// TIA Portal project "Lab5_Exp1_PunchingMachine" (V16)

(* hardware
DEVICE "S7300/ET200M station_1"  S7-300 station
   slot 0: "Rail_0"  Rail  6ES7 390-1***0-0AA0
   slot 2: "PLC_1"  CPU 317-2 PN/DP  6ES7 317-2EK14-0AB0  V3.2
      slot 2: "PROFINET interface_1"  PN-IO
         slot 1: "Port_1"  Port
         slot 2: "Port_2"  Port
*)

// ===== PLC "PLC_1"  CPU 317-2 PN/DP =====

VAR_GLOBAL   // PLC tag table "Default tag table"
   "diStartB" AT %I0.1 : Bool;
   "diGuardDown" AT %I0.2 : Bool;
   "diPunchUp" AT %I0.3 : Bool;
   "diPunchDown" AT %I0.4 : Bool;
   "diStopB" AT %I0.5 : Bool;
   "doPunchDown" AT %Q0.0 : Bool;
   "doReadyIndicator" AT %Q0.1 : Bool;
   "doGDIndicator" AT %Q0.3 : Bool;
   "doGuardDown" AT %Q0.4 : Bool;
   "tvDelayT1" AT %QW66 : Word;
   "tvDelayT2" AT %QW68 : Word;
   "mS_Stop" AT %M100.0 : Bool;
   "mS_GuardDown" AT %M100.1 : Bool;
   "mS_PunchDown" AT %M100.2 : Bool;
   "mS_DelayT1" AT %M100.3 : Bool;
   "mS_GuardUp" AT %M100.4 : Bool;
   "mS_PunchUp" AT %M100.5 : Bool;
   "mT1Elapsed" AT %M100.6 : Bool;
   "mT2Elapsed" AT %M100.7 : Bool;
   "DelayT1" AT %T1 : Timer;
   "DelayT2" AT %T2 : Timer;
   "Tag_1" AT %M200.0 : Bool;
END_VAR

ORGANIZATION_BLOCK "Main"   // OB1, LAD
TITLE = "Main Program Sweep (Cycle)"
{ S7_Optimized_Access := 'FALSE' }
VERSION : 0.1
   VAR_TEMP
      OB1_EV_CLASS : Byte;   // Bits 0-3 = 1 (Coming event), Bits 4-7 = 1 (Event class 1)
      OB1_SCAN_1 : Byte;   // 1 (Cold restart scan 1 of OB 1), 3 (Scan 2-n of OB 1)
      OB1_PRIORITY : Byte;   // Priority of OB Execution
      OB1_OB_NUMBR : Byte;   // 1 (Organization block 1, OB1)
      OB1_RESERVED_1 : Byte;   // Reserved for system
      OB1_RESERVED_2 : Byte;   // Reserved for system
      OB1_PREV_CYCLE : Int;   // Cycle time of previous OB1 scan (milliseconds)
      OB1_MIN_CYCLE : Int;   // Minimum cycle time of OB1 (milliseconds)
      OB1_MAX_CYCLE : Int;   // Maximum cycle time of OB1 (milliseconds)
      OB1_DATE_TIME : Date_And_Time;   // Date and time OB1 started
   END_VAR
   VAR_TEMP   // added for the SCL form of the ladder/FBD networks
      _w1 : Bool;
      _s5time1 : S5Time;
   END_VAR
BEGIN

REGION Network 1: Setting mS_Stop
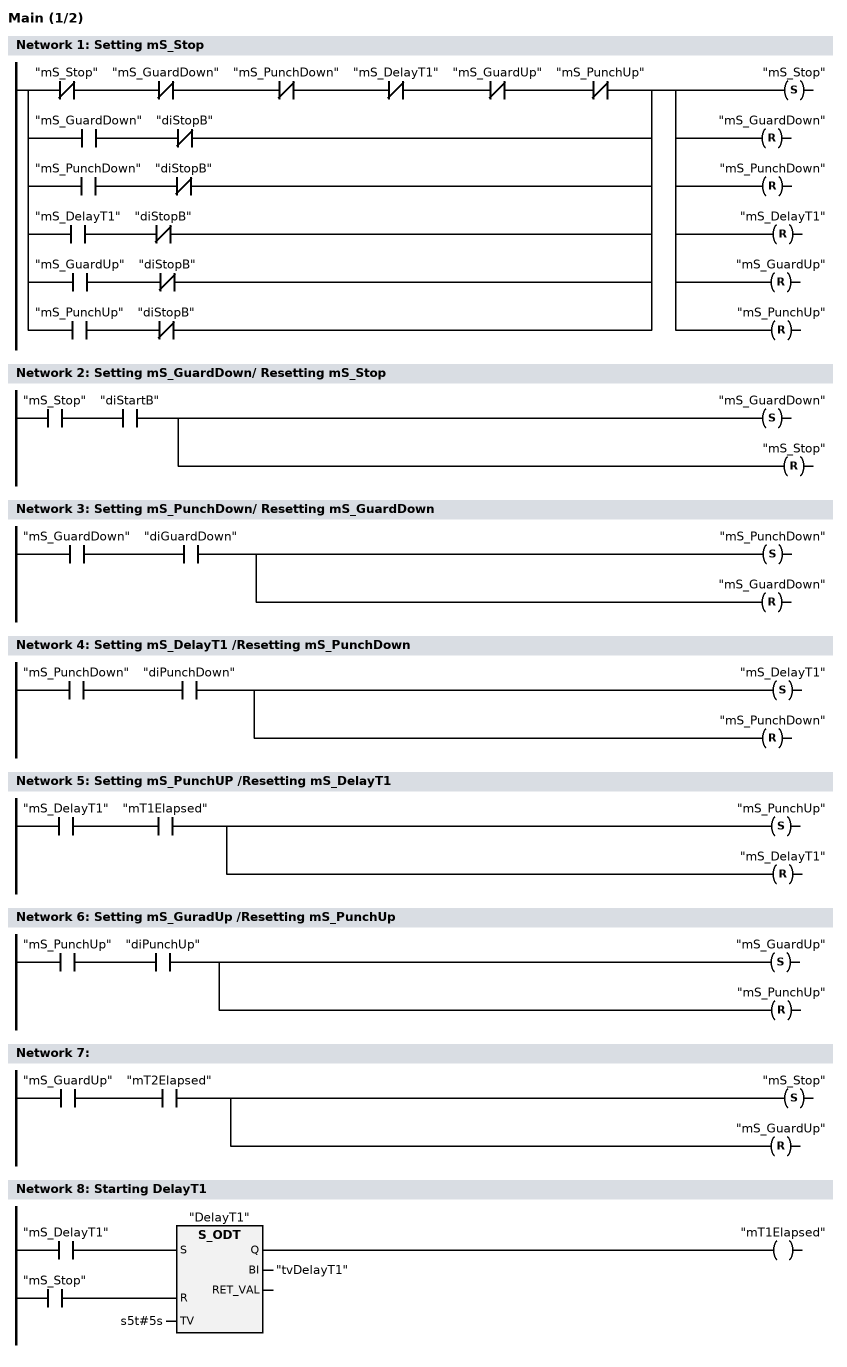
   RUNG wire#powerrail
      I_Contact( "mS_Stop" )
      I_Contact( "mS_GuardDown" )
      I_Contact( "mS_PunchDown" )
      I_Contact( "mS_DelayT1" )
      I_Contact( "mS_GuardUp" )
      I_Contact( "mS_PunchUp" )
      wire#w1
      S_Coil( "mS_Stop" )
   END_RUNG
   RUNG wire#powerrail
      Contact( "mS_GuardDown" )
      I_Contact( "diStopB" )
   END_RUNG wire#w1
   RUNG wire#powerrail
      Contact( "mS_PunchDown" )
      I_Contact( "diStopB" )
   END_RUNG wire#w1
   RUNG wire#powerrail
      Contact( "mS_DelayT1" )
      I_Contact( "diStopB" )
   END_RUNG wire#w1
   RUNG wire#powerrail
      Contact( "mS_GuardUp" )
      I_Contact( "diStopB" )
   END_RUNG wire#w1
   RUNG wire#powerrail
      Contact( "mS_PunchUp" )
      I_Contact( "diStopB" )
   END_RUNG wire#w1
   RUNG wire#w1
      R_Coil( "mS_GuardDown" )
   END_RUNG
   RUNG wire#w1
      R_Coil( "mS_PunchDown" )
   END_RUNG
   RUNG wire#w1
      R_Coil( "mS_DelayT1" )
   END_RUNG
   RUNG wire#w1
      R_Coil( "mS_GuardUp" )
   END_RUNG
   RUNG wire#w1
      R_Coil( "mS_PunchUp" )
   END_RUNG
   // the same network as SCL:
   #_w1 := (NOT "mS_Stop" AND NOT "mS_GuardDown" AND NOT "mS_PunchDown" AND NOT "mS_DelayT1" AND NOT "mS_GuardUp" AND NOT "mS_PunchUp") OR ("mS_GuardDown" AND NOT "diStopB") OR ("mS_PunchDown" AND NOT "diStopB") OR ("mS_DelayT1" AND NOT "diStopB") OR ("mS_GuardUp" AND NOT "diStopB") OR ("mS_PunchUp" AND NOT "diStopB");
   IF #_w1 THEN
       "mS_Stop" := TRUE;
       "mS_GuardDown" := FALSE;
       "mS_PunchDown" := FALSE;
       "mS_DelayT1" := FALSE;
       "mS_GuardUp" := FALSE;
       "mS_PunchUp" := FALSE;
   END_IF;
END_REGION

REGION Network 2: Setting mS_GuardDown/ Resetting mS_Stop
   RUNG wire#powerrail
      Contact( "mS_Stop" )
      Contact( "diStartB" )
      wire#w1
      S_Coil( "mS_GuardDown" )
   END_RUNG
   RUNG wire#w1
      R_Coil( "mS_Stop" )
   END_RUNG
   // the same network as SCL:
   IF "mS_Stop" AND "diStartB" THEN
       "mS_GuardDown" := TRUE;
       "mS_Stop" := FALSE;
   END_IF;
END_REGION

REGION Network 3: Setting mS_PunchDown/ Resetting mS_GuardDown
   RUNG wire#powerrail
      Contact( "mS_GuardDown" )
      Contact( "diGuardDown" )
      wire#w1
      S_Coil( "mS_PunchDown" )
   END_RUNG
   RUNG wire#w1
      R_Coil( "mS_GuardDown" )
   END_RUNG
   // the same network as SCL:
   IF "mS_GuardDown" AND "diGuardDown" THEN
       "mS_PunchDown" := TRUE;
       "mS_GuardDown" := FALSE;
   END_IF;
END_REGION

REGION Network 4: Setting mS_DelayT1 /Resetting mS_PunchDown
   RUNG wire#powerrail
      Contact( "mS_PunchDown" )
      Contact( "diPunchDown" )
      wire#w1
      S_Coil( "mS_DelayT1" )
   END_RUNG
   RUNG wire#w1
      R_Coil( "mS_PunchDown" )
   END_RUNG
   // the same network as SCL:
   IF "mS_PunchDown" AND "diPunchDown" THEN
       "mS_DelayT1" := TRUE;
       "mS_PunchDown" := FALSE;
   END_IF;
END_REGION

REGION Network 5: Setting mS_PunchUP /Resetting mS_DelayT1
   RUNG wire#powerrail
      Contact( "mS_DelayT1" )
      Contact( "mT1Elapsed" )
      wire#w1
      S_Coil( "mS_PunchUp" )
   END_RUNG
   RUNG wire#w1
      R_Coil( "mS_DelayT1" )
   END_RUNG
   // the same network as SCL:
   IF "mS_DelayT1" AND "mT1Elapsed" THEN
       "mS_PunchUp" := TRUE;
       "mS_DelayT1" := FALSE;
   END_IF;
END_REGION

REGION Network 6: Setting mS_GuradUp /Resetting mS_PunchUp
   RUNG wire#powerrail
      Contact( "mS_PunchUp" )
      Contact( "diPunchUp" )
      wire#w1
      S_Coil( "mS_GuardUp" )
   END_RUNG
   RUNG wire#w1
      R_Coil( "mS_PunchUp" )
   END_RUNG
   // the same network as SCL:
   IF "mS_PunchUp" AND "diPunchUp" THEN
       "mS_GuardUp" := TRUE;
       "mS_PunchUp" := FALSE;
   END_IF;
END_REGION

REGION Network 7
   RUNG wire#powerrail
      Contact( "mS_GuardUp" )
      Contact( "mT2Elapsed" )
      wire#w1
      S_Coil( "mS_Stop" )
   END_RUNG
   RUNG wire#w1
      R_Coil( "mS_GuardUp" )
   END_RUNG
   // the same network as SCL:
   IF "mS_GuardUp" AND "mT2Elapsed" THEN
       "mS_Stop" := TRUE;
       "mS_GuardUp" := FALSE;
   END_IF;
END_REGION

REGION Network 8: Starting DelayT1
   RUNG wire#powerrail
      Contact( "mS_DelayT1" )
      S_ODT(T_NO := "DelayT1", R := wire#w1, TV := s5t#5s, BI => "tvDelayT1", RET_VAL =>)
      Coil( "mT1Elapsed" )
   END_RUNG
   RUNG wire#powerrail
      Contact( "mS_Stop" )
   END_RUNG wire#w1
   // the same network as SCL:
   #_s5time1 := S_ODT(T_NO := "DelayT1",
                      S := "mS_DelayT1",
                      R := "mS_Stop",
                      TV := s5t#5s,
                      Q => #_w1,
                      BI => "tvDelayT1");
   "mT1Elapsed" := #_w1;
END_REGION

REGION Network 9: Starting DelayT2
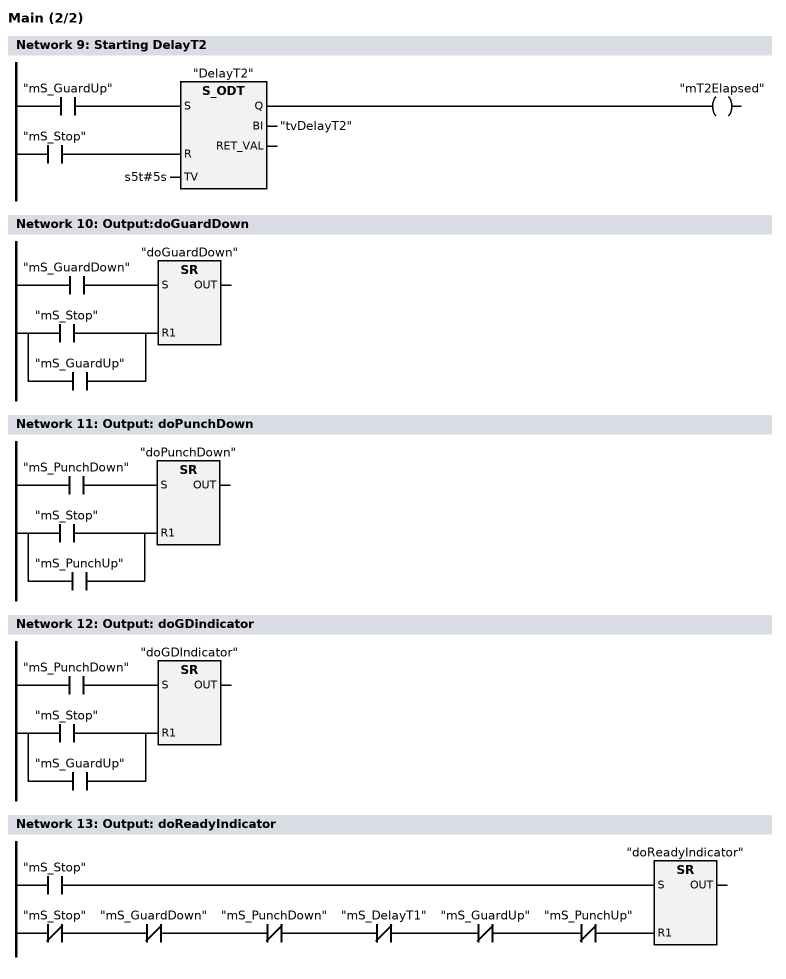
   RUNG wire#powerrail
      Contact( "mS_GuardUp" )
      S_ODT(T_NO := "DelayT2", R := wire#w1, TV := s5t#5s, BI => "tvDelayT2", RET_VAL =>)
      Coil( "mT2Elapsed" )
   END_RUNG
   RUNG wire#powerrail
      Contact( "mS_Stop" )
   END_RUNG wire#w1
   // the same network as SCL:
   #_s5time1 := S_ODT(T_NO := "DelayT2",
                      S := "mS_GuardUp",
                      R := "mS_Stop",
                      TV := s5t#5s,
                      Q => #_w1,
                      BI => "tvDelayT2");
   "mT2Elapsed" := #_w1;
END_REGION

REGION Network 10: Output:doGuardDown
   RUNG wire#powerrail
      Contact( "mS_GuardDown" )
      S_SR(operand := "doGuardDown", r1 := wire#w1)
   END_RUNG
   RUNG wire#powerrail
      Contact( "mS_Stop" )
   END_RUNG wire#w1
   RUNG wire#powerrail
      Contact( "mS_GuardUp" )
   END_RUNG wire#w1
   // the same network as SCL:
   IF "mS_GuardDown" THEN
       "doGuardDown" := TRUE;   // SR flip-flop
   END_IF;
   IF "mS_Stop" OR "mS_GuardUp" THEN "doGuardDown" := FALSE; END_IF;
END_REGION

REGION Network 11: Output: doPunchDown
   RUNG wire#powerrail
      Contact( "mS_PunchDown" )
      S_SR(operand := "doPunchDown", r1 := wire#w1)
   END_RUNG
   RUNG wire#powerrail
      Contact( "mS_Stop" )
   END_RUNG wire#w1
   RUNG wire#powerrail
      Contact( "mS_PunchUp" )
   END_RUNG wire#w1
   // the same network as SCL:
   IF "mS_PunchDown" THEN
       "doPunchDown" := TRUE;   // SR flip-flop
   END_IF;
   IF "mS_Stop" OR "mS_PunchUp" THEN "doPunchDown" := FALSE; END_IF;
END_REGION

REGION Network 12: Output: doGDindicator
   RUNG wire#powerrail
      Contact( "mS_PunchDown" )
      S_SR(operand := "doGDIndicator", r1 := wire#w1)
   END_RUNG
   RUNG wire#powerrail
      Contact( "mS_Stop" )
   END_RUNG wire#w1
   RUNG wire#powerrail
      Contact( "mS_GuardUp" )
   END_RUNG wire#w1
   // the same network as SCL:
   IF "mS_PunchDown" THEN
       "doGDIndicator" := TRUE;   // SR flip-flop
   END_IF;
   IF "mS_Stop" OR "mS_GuardUp" THEN "doGDIndicator" := FALSE; END_IF;
END_REGION

REGION Network 13: Output: doReadyIndicator
   RUNG wire#powerrail
      Contact( "mS_Stop" )
      S_SR(operand := "doReadyIndicator", r1 := wire#w1)
   END_RUNG
   RUNG wire#powerrail
      I_Contact( "mS_Stop" )
      I_Contact( "mS_GuardDown" )
      I_Contact( "mS_PunchDown" )
      I_Contact( "mS_DelayT1" )
      I_Contact( "mS_GuardUp" )
      I_Contact( "mS_PunchUp" )
   END_RUNG wire#w1
   // the same network as SCL:
   IF "mS_Stop" THEN
       "doReadyIndicator" := TRUE;   // SR flip-flop
   END_IF;
   IF NOT "mS_Stop" AND NOT "mS_GuardDown" AND NOT "mS_PunchDown" AND NOT "mS_DelayT1" AND NOT "mS_GuardUp" AND NOT "mS_PunchUp" THEN
       "doReadyIndicator" := FALSE;
   END_IF;
END_REGION
END_ORGANIZATION_BLOCK